// TwinCAT 3 PLC project mobject_types
// Title: mobject-types
// Company: mobject
// Author: mobject dev team
// ProjectVersion: 0.1.0
// ProgramVersion: 3.1.4024.0
// libraries:
//   mobject-collections,1.1.0,mobject
//   mobject-deserialization,0.1.0,mobject
//   mobject-disposable,1.0.0,mobject
//   mobject-enumerable,1.1.0,mobject
//   mobject-serialization,0.4.0,mobject
//   Tc2_System, * (Beckhoff Automation GmbH)
//   Tc2_Utilities, * (Beckhoff Automation GmbH)
// project tree:
//   DatatypePacks/ PlcBasicDatatypePack.TcPOU
//   Datatypes/ Datatypes.TcPOU (not stored)
//   Datatype/Alias/ _HRESULT.TcPOU (not stored), _FLOAT.TcPOU
//   Datatype/Primitive/ _BOOL.TcPOU (not stored), _BYTE.TcPOU (not stored), _DINT.TcPOU (not stored), _TIME_OF_DAY.TcPOU (not stored), _REAL.TcPOU (not stored), _LWORD.TcPOU (not stored), _INT.TcPOU (not stored), _LINT.TcPOU (not stored), _LREAL.TcPOU (not stored), _SINT.TcPOU (not stored), _TOD.TcPOU (not stored), _DT.TcPOU (not stored), _UINT.TcPOU (not stored), _USINT.TcPOU (not stored), _UDINT.TcPOU (not stored), _ULINT.TcPOU (not stored), _WORD.TcPOU (not stored), _DWORD.TcPOU (not stored)
//   Datatype/Structs/ _TIMESTRUCT.TcPOU (not stored)
//   Interfaces/ I_Datatype.TcIO (not stored), I_DatatypePack.TcIO (not stored), I_Datatypes.TcIO (not stored), I_StructuredDatatype.TcIO (not stored), I_AliasDatatype.TcIO (not stored)
//   _Internal/DatatypeVisitor/ I_DatatypeVisitor.TcIO (not stored)
//   _Internal/Datatype/ AliasDatatypeBase.TcPOU (not stored), DatatypeBase.TcPOU (not stored), StructuredDatatypeBase.TcPOU (not stored)
//   _Internal/MembersHost/ I_HostMembers.TcIO (not stored), MembersHost.TcPOU (not stored)

// ---- DatatypePacks/PlcBasicDatatypePack.TcPOU
{attribute 'linkalways'} 
{attribute 'no_explicit_call' := 'This FB is a CLASS and must be accessed using methods or properties'}
{attribute 'enable_dynamic_creation'}
FUNCTION_BLOCK PlcBasicDatatypePack IMPLEMENTS I_DatatypePack
VAR
	// alias
	_hresult : _HRESULT(0);
    _float : _FLOAT(0);
	
	// primitive
	_bool : _BOOL(FALSE);
	_byte : _BYTE(0);
	_dint : _DINT(0);
	_dt : _DT(DT#1970-1-1-0:0:0);
	_dword : _DWORD(0);
	_int : _INT(0);
	_lint : _LINT(0);
	_lreal : _LREAL(0);
	_lword : _LWORD(0);
	_real : _REAL(0);
	_sint : _SINT(0);
	_time_of_day : _TIME_OF_DAY(TOD#0:0:0);
	_tod : _TOD(TOD#0:0:0);
	_udint : _UDINT(0);
	_uint : _UINT(0);
	_ulint : _ULINT(0);
	_usint : _USINT(0);
	_word : _WORD(0);
	
	// structures
	_timestruct : _TIMESTRUCT();
	
END_VAR

METHOD RegisterWith
VAR_INPUT
	Datatypes : I_Datatypes;
END_VAR
// alias
Datatypes.RegisterDatatype(_hresult);
Datatypes.RegisterDatatype(_float);

// primitive
Datatypes.RegisterDatatype(_bool);
Datatypes.RegisterDatatype(_byte);
Datatypes.RegisterDatatype(_dint);
Datatypes.RegisterDatatype(_dt);
Datatypes.RegisterDatatype(_dword);
Datatypes.RegisterDatatype(_int);
Datatypes.RegisterDatatype(_lint);
Datatypes.RegisterDatatype(_lreal);
Datatypes.RegisterDatatype(_lword);
Datatypes.RegisterDatatype(_real);
Datatypes.RegisterDatatype(_sint);
Datatypes.RegisterDatatype(_time_of_day);
Datatypes.RegisterDatatype(_tod);
Datatypes.RegisterDatatype(_udint);
Datatypes.RegisterDatatype(_uint);
Datatypes.RegisterDatatype(_ulint);
Datatypes.RegisterDatatype(_usint);
Datatypes.RegisterDatatype(_word);

// structures
Datatypes.RegisterDatatype(_timestruct);
END_METHOD

END_FUNCTION_BLOCK

// ---- Datatype/Alias/_FLOAT.TcPOU
{attribute 'linkalways'} 
{attribute 'no_explicit_call' := 'This FB is a CLASS and must be accessed using methods or properties'}
{attribute 'enable_dynamic_creation'}
FUNCTION_BLOCK _FLOAT EXTENDS AliasDatatypeBase
VAR
	localData : FLOAT;
	activeData : REFERENCE TO FLOAT REF= localData;
	aliasBaseType : _LREAL(localData);
END_VAR

PROPERTY PUBLIC Address : PVOID
GET
Address := ADR(activeData);
END_GET
END_PROPERTY

METHOD PUBLIC ClearReference
VAR_INPUT
END_VAR
activeData REF= localData;
SetBaseTypeReference();
END_METHOD

METHOD PUBLIC Clone : I_Datatype
VAR
    pClone : POINTER TO _FLOAT;
END_VAR
pClone := __NEW(_FLOAT(InitialValue := Value));
Clone := pClone^;
END_METHOD

METHOD FB_init : BOOL
VAR_INPUT
	bInitRetains : BOOL; // if TRUE, the retain variables are initialized (warm start / cold start)
	bInCopyCode : BOOL;  // if TRUE, the instance afterwards gets moved into the copy code (online change)
	InitialValue : FLOAT;
END_VAR
localData := InitialValue;
SetBaseTypeReference();
AddBaseType(aliasBaseType);
END_METHOD

PROPERTY PUBLIC Identifier : T_MAXSTRING
GET
Identifier := 'FLOAT';
END_GET
END_PROPERTY

METHOD PUBLIC MakeReferenceTo
VAR_INPUT
	ReferenceTarget : REFERENCE TO FLOAT;
END_VAR
activeData REF= ReferenceTarget;
SetBaseTypeReference();
END_METHOD

METHOD PROTECTED SetBaseTypeReference
VAR_INPUT
END_VAR
aliasBaseType.MakeReferenceTo(activeData);
END_METHOD

PROPERTY PUBLIC Size : UDINT
GET
Size := SIZEOF(activeData);
END_GET
END_PROPERTY

METHOD TryMakeReferenceTo : BOOL
VAR_INPUT
	Target : I_Datatype;
END_VAR
VAR
	pTargetData : POINTER TO FLOAT;
END_VAR
IF NOT (Target.IecType = IecType) THEN
	RETURN;
END_IF

pTargetData := Target.Address;
activeData REF= pTargetData^;
SetBaseTypeReference();
TryMakeReferenceTo := TRUE;
END_METHOD

PROPERTY PUBLIC Value : FLOAT
GET
Value := activeData;
END_GET
SET
activeData := Value;
END_SET
END_PROPERTY

END_FUNCTION_BLOCK
